VAR_GLOBAL
	var01		:	INT;
END_VAR

(* stored: Version 1.1.0.1, ProductVersion 3.1.4020.6
   GVL GVL01: Id {666e17ed-9ecf-47c0-bf89-64f688967938} *)
